TYPE TFCodiciPerFormatura :
STRUCT
	Code : ARRAY[1..MAXFORMINGCODE] OF INT;
END_STRUCT
END_TYPE

(* stored: Version 1.1.0.1, ProductVersion 3.1.4024.9
   DUT TFCodiciPerFormatura: Id {184eb9e1-85e7-41a3-a7e4-c79f0ce22d62} *)
